// Interface for indicating that an object is for detecting the change of some object/value.
INTERFACE I_ChangeDetector EXTENDS __SYSTEM.IQueryInterface

// Indicates if the object has changed.
// [get] Returns flag indicating of object has changed.
PROPERTY HasChanged : BOOL
GET
END_GET
END_PROPERTY

END_INTERFACE

(* stored: Version 1.1.0.1
   Itf I_ChangeDetector: Id {69563f31-3a03-0f75-1bd5-63482cbbb489}
   Property HasChanged: Id {8b88e136-4add-0ad9-2874-091307727d57}
   Get Get: Id {f713254a-f4c0-0594-2bda-027754937f11} *)
